FUNCTION_BLOCK Sensor_Bool (* Basic Function Block Type *)
  (* Standard: 61499-2 *)
  (* Version 0.0, 2/2/2026, Schneider Electric, Template *)
  PACKAGE Main;
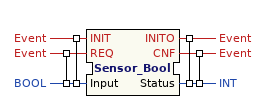
  EVENT_INPUT
    INIT WITH Input; (* Initialization Request *)
    REQ WITH Input; (* Normal Execution Request *)
  END_EVENT
  EVENT_OUTPUT
    INITO WITH Status; (* Initialization Confirm *)
    CNF WITH Status; (* Execution Confirmation *)
  END_EVENT
  VAR_INPUT
    Input : BOOL; (* Input event qualifier *)
  END_VAR
  VAR_OUTPUT
    Status : INT; (* Output event qualifier *)
  END_VAR
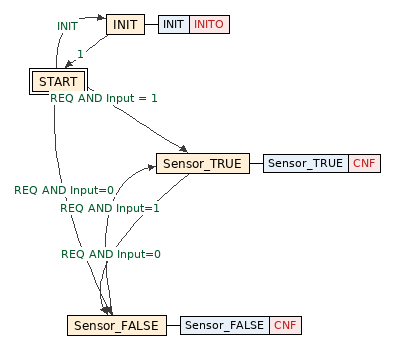
  EC_STATES
    START; (* Initial State *)
    INIT : INIT -> INITO; (* Initialization *)
    Sensor_TRUE : Sensor_TRUE -> CNF; (* Normal execution *)
    Sensor_FALSE : Sensor_FALSE -> CNF; (* Normal execution *)
  END_STATES
  EC_TRANSITIONS
    START TO INIT := INIT;
    INIT TO START := 1;
    START TO Sensor_TRUE := REQ AND Input = 1;
    Sensor_TRUE TO Sensor_FALSE := REQ AND Input=0;
    START TO Sensor_FALSE := REQ AND Input=0;
    Sensor_FALSE TO Sensor_TRUE := REQ AND Input=1;
  END_TRANSITIONS
  ALGORITHM INIT IN ST: (* Initialization algorithm *)
;
  END_ALGORITHM
  ALGORITHM Sensor_TRUE IN ST: (* Normally executed algorithm *)
Status := 1;
  END_ALGORITHM
  ALGORITHM Sensor_FALSE IN ST:
Status:= 0;
  END_ALGORITHM
END_FUNCTION_BLOCK
